FUNCTION_BLOCK AUDI_FIELDBUS_UDINT_TO_SIGNAL (* Mirrors IN->OUT if Signal Valid. *)
  (* Standard: 61499-1; Description: Copyright (c) 2026 HR Agrartechnik GmbH This program and the accompanying materials are made available under the terms of the Eclipse Public License 2.0 which is available at https://www.eclipse.org/legal/epl-2.0/ SPDX-License-Identifier: EPL-2.0 *)
  (* Version 1.0, 2026-05-31, Franz Höpfinger, HR Agrartechnik GmbH *)
  PACKAGE logiBUS::signalprocessing::fieldbus;
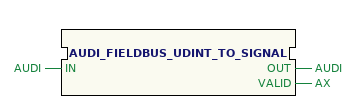
  SOCKETS
    IN : adapter::types::unidirectional::AUDI; (* Input *)
  END_SOCKETS
  PLUGS
    OUT : adapter::types::unidirectional::AUDI; (* Output Filtered *)
    VALID : adapter::types::unidirectional::AX; (* TRUE if Signal is VALID *)
  END_PLUGS
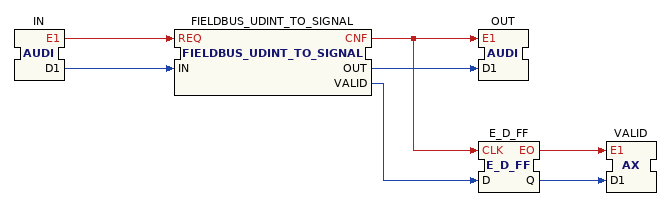
  FBS
    FIELDBUS_UDINT_TO_SIGNAL : logiBUS::signalprocessing::fieldbus::FIELDBUS_UDINT_TO_SIGNAL;
    E_D_FF : iec61499::events::E_D_FF;
  END_FBS
  EVENT_CONNECTIONS
    IN.E1 TO FIELDBUS_UDINT_TO_SIGNAL.REQ;
    FIELDBUS_UDINT_TO_SIGNAL.CNF TO OUT.E1;
    FIELDBUS_UDINT_TO_SIGNAL.CNF TO E_D_FF.CLK;
    E_D_FF.EO TO VALID.E1;
  END_CONNECTIONS
  DATA_CONNECTIONS
    IN.D1 TO FIELDBUS_UDINT_TO_SIGNAL.IN;
    FIELDBUS_UDINT_TO_SIGNAL.OUT TO OUT.D1;
    FIELDBUS_UDINT_TO_SIGNAL.VALID TO E_D_FF.D;
    E_D_FF.Q TO VALID.D1;
  END_CONNECTIONS
END_FUNCTION_BLOCK
